PROGRAM DatabaseRecord
VAR
	tTimeout: TIME := T#5s;
	bExecute: BOOL;
	nState: INT;
	
	fbFormatString: FB_FormatString;
	fbDBRecordSelect: FB_DBRecordArraySelect;
	
	timer: TON := (IN:= TRUE);
END_VAR

(*------ Add data to database every tStoreVar time ------*)
timer(IN:= , PT:= tStoreVar, Q=> , ET=> );

fbDBRecordSelect(
	sNetID:= , 
	hDBID:= 1, 
	pCmdAddr:= , 
	cbCmdSize:= , 
	nStartIndex:= 0, 
	nRecordCount:= 1, 
	pDestAddr:= ADR(nID), 
	cbRecordArraySize:= SIZEOF(nID), 
	bExecute:= , 
	tTimeout:= tTimeout);

fbFormatString(
		sFormat:= 'INSERT INTO [myTable] ([Timestamp],[Temperature1],[Temperature2],[Temperature3], [Status], [Comment]) OUTPUT INSERTED.ID VALUES(CURRENT_TIMESTAMP,%0.5f,%0.5f,%0.5f,%d,$'%s$');',  
		arg1:= F_REAL(rTemp1),
		arg2:= F_REAL(rTemp2),
		arg3:= F_REAL(rTemp3),
		arg4:= F_INT(bToggle),
		arg5:= F_STRING(sComment));
(*
//FORMAT FOR MYSQL 
fbFormatString(
		sFormat:= 'INSERT INTO myTable (Timestamp,Temperature1,Temperature2,Temperature3, Status, Comment) VALUES(CURRENT_TIMESTAMP,%0.5f,%0.5f,%0.5f,%d,$'%s$'); SELECT LAST_INSERT_ID();',  
		arg1:= F_REAL(rTemp1),
		arg2:= F_REAL(rTemp2),
		arg3:= F_REAL(rTemp3),
		arg4:= F_INT(bToggle),
		arg5:= F_STRING(sComment));
*)

(*
//FORMAT FOR SQLite 
fbFormatString(
		sFormat:= 'INSERT INTO [myTable] ([Timestamp],[Temperature1],[Temperature2],[Temperature3], [Status], [Comment]) VALUES(CURRENT_TIMESTAMP,%0.5f,%0.5f,%0.5f,%d,$'%s$'); SELECT LAST_INSERT_ROWID();',  
		arg1:= F_REAL(rTemp1),
		arg2:= F_REAL(rTemp2),
		arg3:= F_REAL(rTemp3),
		arg4:= F_INT(bToggle),
		arg5:= F_STRING(sComment));
*)

CASE nState OF 
	0:
	IF NOT fbFormatString.bError AND fbFormatString.sOut <> '' THEN
		nState := 10;
	END_IF

	10:
	IF timer.Q THEN
		fbDBRecordSelect.pCmdAddr := ADR(fbFormatString.sOut);
		fbDBRecordSelect.cbCmdSize := SIZEOF(fbFormatString.sOut);
		fbDBRecordSelect.bExecute := TRUE;
		timer.IN := FALSE;
		nState := 20;
	END_IF

	20:
	IF NOT fbDBRecordSelect.bBusy AND NOT fbDBRecordSelect.bError THEN
		fbDBRecordSelect.bExecute := FALSE;
		timer.IN := TRUE;
		nState := 0;
	END_IF
END_CASE

END_PROGRAM

(* stored: Version 1.1.0.1, ProductVersion 3.1.4020.12
   POU DatabaseRecord: Id {9d9db9b5-050c-405c-86b5-723f1f75410c}, SpecialFunc None *)
